KUKA KRL data list: kukavarproxyvelperc.dat

&ACCESS RVP
&REL 1
&PARAM TEMPLATE = C:\KRC\Roboter\Template\vorgabe
&PARAM EDITMASK = *
DEFDAT kukavarproxyvelperc
;FOLD EXTERNAL DECLARATIONS;%{PE}%MKUKATPBASIS,%CEXT,%VCOMMON,%P
;FOLD BASISTECH EXT;%{PE}%MKUKATPBASIS,%CEXT,%VEXT,%P
EXT  BAS (BAS_COMMAND  :IN,REAL  :IN )
DECL INT SUCCESS
;ENDFOLD (BASISTECH EXT)
;FOLD USER EXT;%{E}%MKUKATPUSER,%CEXT,%VEXT,%P
;Make here your modifications
STRUC AXISVELPERC_TYP INT A1, A2, A3, A4, A5, A6
STRUC EXTAXVELPERC_TYP INT E1, E2, E3
STRUC AXISFBSET_TYP E6AXIS AXIS_SET, AXISVELPERC_TYP AXIS_VEL_SET, EXTAXVELPERC_TYP EXTAX_VEL_SET
DECL AXISFBSET_TYP AXIS_FB_SET
;ENDFOLD (USER EXT)
;ENDFOLD (EXTERNAL DECLERATIONS)
ENDDAT
